FUNCTION_BLOCK "Filter_1_sleeve"
{ S7_Optimized_Access := 'TRUE' }
VERSION : 0.1
   VAR_IN_OUT
      filter : "UDT_Filter_1_sleeve";
   END_VAR

   VAR
      first_scan { ExternalAccessible := 'False'; ExternalVisible := 'False'; ExternalWritable := 'False'} : Bool;   // Indicate if first scan for initialization
      desired_open_command { ExternalAccessible := 'False'; ExternalVisible := 'False'; ExternalWritable := 'False'} : Bool;   // Actual desired command based on active mode
      validated_open_command { ExternalAccessible := 'False'; ExternalVisible := 'False'; ExternalWritable := 'False'} : Bool;   // Desired command if not interlocked
      pulse_timer {InstructionName := 'TON_TIME'; LibVersion := '1.0'; ExternalAccessible := 'False'; ExternalVisible := 'False'; ExternalWritable := 'False'; S7_SetPoint := 'False'} : TON_TIME;   // Timer for pulse active
      interval_timer {InstructionName := 'TON_TIME'; LibVersion := '1.0'; ExternalAccessible := 'False'; ExternalVisible := 'False'; ExternalWritable := 'False'; S7_SetPoint := 'False'} : TON_TIME;   // Timer between pulses
      fb_XY { ExternalWritable := 'False'; S7_SetPoint := 'False'} : "Solenoid_valve";
   END_VAR

   VAR CONSTANT
      IDLE : Int := 1;   // Filter in idle state
      WAITING : Int := 2;   // Filter waiting for next pulse
      ACTIVE : Int := 3;   // Filter pulsing air
   END_VAR


BEGIN
	REGION Initialization
	    IF #first_scan THEN
	        #first_scan := FALSE;
	        #filter.STATUS.state := #IDLE;
	    END_IF;
	END_REGION

	REGION Map internal valves
	    #fb_XY(#filter.DEVICES.XY);
	END_REGION

	REGION Determine desired target
	    IF #filter.CMD.manual_mode THEN
	        #desired_open_command := #filter.CMD.manual;
	    ELSE
	        #desired_open_command := #filter.CMD.auto;
	    END_IF;
	    // Only update validated command if not interlocked
	    IF NOT #filter.CMD.interlocked THEN
	        #validated_open_command := #desired_open_command;
	    END_IF;
	    // If interlocked, validated_open_command retains its last value
	END_REGION

	REGION Timers
	    #interval_timer(IN := (#filter.STATUS.state = #WAITING),
	                    PT := #filter.SETTING.interval_duration);

	    #pulse_timer(IN := (#filter.STATUS.state = #ACTIVE),
	                 PT := #filter.SETTING.pulse_duration);
	END_REGION

	REGION FSM logic
	    CASE #filter.STATUS.state OF
	        #IDLE:
	            IF #desired_open_command THEN
	                #filter.STATUS.state := #ACTIVE;
	            END_IF;

	        #WAITING:
	            IF #interval_timer.Q THEN
	                IF #desired_open_command THEN
	                    #filter.STATUS.state := #ACTIVE;
	                ELSE
	                    #filter.STATUS.state := #IDLE;
	                END_IF;
	            ELSIF NOT #desired_open_command THEN
	                #filter.STATUS.state := #IDLE; // return to idle if command removed
	            END_IF;

	        #ACTIVE:
	            IF #pulse_timer.Q THEN
	                #filter.STATUS.state := #WAITING;
	            ELSIF NOT #desired_open_command THEN
	                #filter.STATUS.state := #IDLE; // return to idle if command removed
	            END_IF;

	        ELSE: // Safety fallback
	            #filter.STATUS.state := #IDLE;
	    END_CASE;
	END_REGION

	REGION Output mapping
	    #filter.DEVICES.XY.CMD.auto := FALSE;
	    #filter.STATUS.is_idle := FALSE;
	    #filter.STATUS.is_waiting := FALSE;
	    #filter.STATUS.is_active := FALSE;

	    CASE #filter.STATUS.state OF
	        #IDLE:
	            #filter.STATUS.is_idle := TRUE;

	        #WAITING:
	            #filter.STATUS.is_waiting := TRUE;

	        #ACTIVE:
	            #filter.DEVICES.XY.CMD.auto := TRUE;
	            #filter.STATUS.is_active := TRUE;
	    END_CASE;
	END_REGION
END_FUNCTION_BLOCK

